FUNCTION_BLOCK T_ComponentsInitialisedSuccess EXTENDS T_UnitTestBase
VAR
  list : T_ComponentsCollection(10);
  newComponent, newComponent2 : T_ComponentMock; 
  actual1, actual2 : BOOL;
END_VAR

// Arrange
list.AddComponent(newComponent);
list.AddComponent(newComponent2);

//Act
list.CyclicLogic();

//Assert
actual1 := list.AllInitialised();

assertion.AssertEquals_BOOL(TRUE, actual1, 'actual1 := list.AllInitialised();');
TestFinished();

END_FUNCTION_BLOCK

(* stored: Version 1.1.0.1, ProductVersion 3.1.4024.12
   POU T_ComponentsInitialisedSuccess: Id {94c45123-908a-477f-9d80-ff0f93786fcc}, SpecialFunc None *)
